PROGRAM Read_Strain
VAR
	Strain_Left		: REAL;
	Strain_Right	: REAL;
	
	nBit_Left AT %I*	: INT;
	nBit_Right AT %I*	: INT;
END_VAR

(* convert to strain *)
Strain_Left	:= ((nBit_Left/32767)*1090)+10;
Strain_Right := ((nBit_Right/32767)*1090)+10;

END_PROGRAM

(* stored: Version 1.1.0.1, ProductVersion 3.1.4024.6
   POU Read_Strain: Id {16e1bd7e-c7ed-4e20-b439-b4719d1dd6a8}, SpecialFunc None *)
